{attribute addProperty BoxType "EL6861-0000-0016"}
{attribute addProperty Id "COM_TxPDO_Map_InputsAT %I*COM_TxPDO_Map_Inputs_73F0C8F110401300COM_RxPDO_MapAT %Q*COM_RxPDO_Map_3D77FD3410401300WcStateAT %I*WcState_98A4DF7520.250InfoDataAT %I*InfoData_BC63D37F80100"}
{attribute addProperty CRC "943410007"}
{attribute addProperty SizeInBites "2162"}
{attribute addProperty SizeInBytes "270.25"}
TYPE EL6861_B662EC3C :
STRUCT
	{attribute addProperty Name "COM_TxPDO_Map_Inputs"}
	COM_TxPDO_Map_Inputs : COM_TxPDO_Map_Inputs_73F0C8F1;
	{attribute addProperty Name "COM_RxPDO_Map"}
	COM_RxPDO_Map : COM_RxPDO_Map_3D77FD34;
	{attribute addProperty Name "WcState"}
	WcState : WcState_98A4DF75;
	{attribute addProperty Name "InfoData"}
	InfoData : InfoData_BC63D37F;
END_STRUCT
END_TYPE

(* stored: Version 1.2.0.0, ProductVersion 3.1.4024.9
   DUT EL6861_B662EC3C: Id {eb9bfd14-51d7-4360-84fe-6ab7a89dcc1a} *)
